TYPE udt_SRxx_Input_Image :
STRUCT
	Retry : BOOL;
	Bypass :BOOL;
END_STRUCT
END_TYPE

(* stored: Version 1.1.0.1, ProductVersion 3.1.4024.12
   DUT udt_SRxx_Input_Image: Id {d95db831-f0ce-43ed-8744-7e6bbc60c015} *)
